Xinje XDPPro project, PLC1: XDC-32 (software 3.8.1a 2026-04-22)

PROGRAM 梯形图

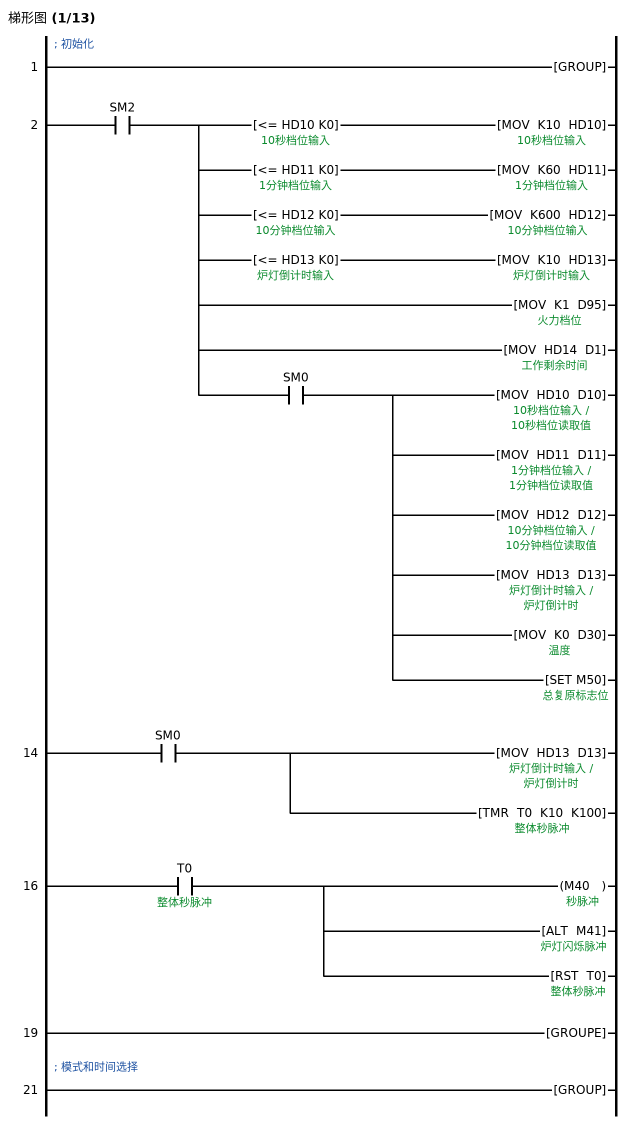
; 初始化
GROUP
LD     SM2
MPS
AND<=  HD10 K0	; 10秒档位输入
MOV    K10 HD10	; 10秒档位输入
MRD
AND<=  HD11 K0	; 1分钟档位输入
MOV    K60 HD11	; 1分钟档位输入
MRD
AND<=  HD12 K0	; 10分钟档位输入
MOV    K600 HD12	; 10分钟档位输入
MRD
AND<=  HD13 K0	; 炉灯倒计时输入
MOV    K10 HD13	; 炉灯倒计时输入
MPP
MOV    K1 D95	; 火力档位
MOV    HD14 D1	; 工作剩余时间
AND    SM0
MOV    HD10 D10	; 10秒档位输入 / 10秒档位读取值
MOV    HD11 D11	; 1分钟档位输入 / 1分钟档位读取值
MOV    HD12 D12	; 10分钟档位输入 / 10分钟档位读取值
MOV    HD13 D13	; 炉灯倒计时输入 / 炉灯倒计时
MOV    K0 D30	; 温度
SET    M50	; 总复原标志位
LD     SM0
MOV    HD13 D13	; 炉灯倒计时输入 / 炉灯倒计时
TMR    T0 K10 K100	; 整体秒脉冲
LD     T0	; 整体秒脉冲
OUT    M40	; 秒脉冲
ALT    M41	; 炉灯闪烁脉冲
RST    T0	; 整体秒脉冲
GROUPE
; 模式和时间选择
GROUP

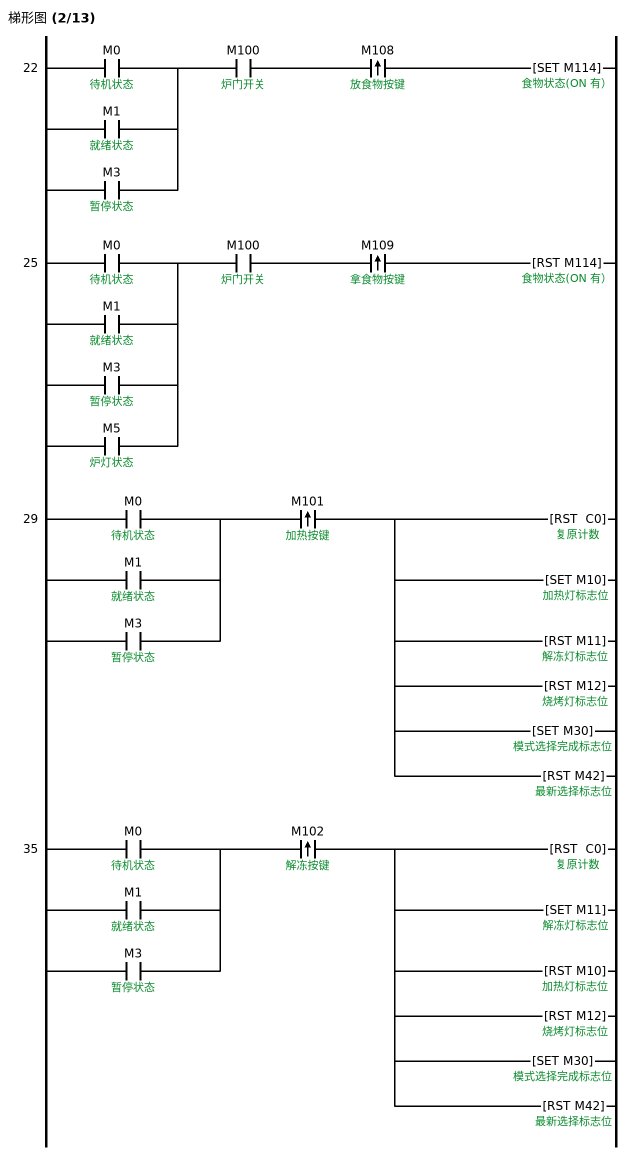
LD     M0	; 待机状态
OR     M1	; 就绪状态
OR     M3	; 暂停状态
AND    M100	; 炉门开关
ANDP   M108	; 放食物按键
SET    M114	; 食物状态(ON 有）
LD     M0	; 待机状态
OR     M1	; 就绪状态
OR     M3	; 暂停状态
OR     M5	; 炉灯状态
AND    M100	; 炉门开关
ANDP   M109	; 拿食物按键
RST    M114	; 食物状态(ON 有）
LD     M0	; 待机状态
OR     M1	; 就绪状态
OR     M3	; 暂停状态
ANDP   M101	; 加热按键
RST    C0	; 复原计数
SET    M10	; 加热灯标志位
RST    M11	; 解冻灯标志位
RST    M12	; 烧烤灯标志位
SET    M30	; 模式选择完成标志位
RST    M42	; 最新选择标志位
LD     M0	; 待机状态
OR     M1	; 就绪状态
OR     M3	; 暂停状态
ANDP   M102	; 解冻按键
RST    C0	; 复原计数
SET    M11	; 解冻灯标志位
RST    M10	; 加热灯标志位
RST    M12	; 烧烤灯标志位
SET    M30	; 模式选择完成标志位
RST    M42	; 最新选择标志位

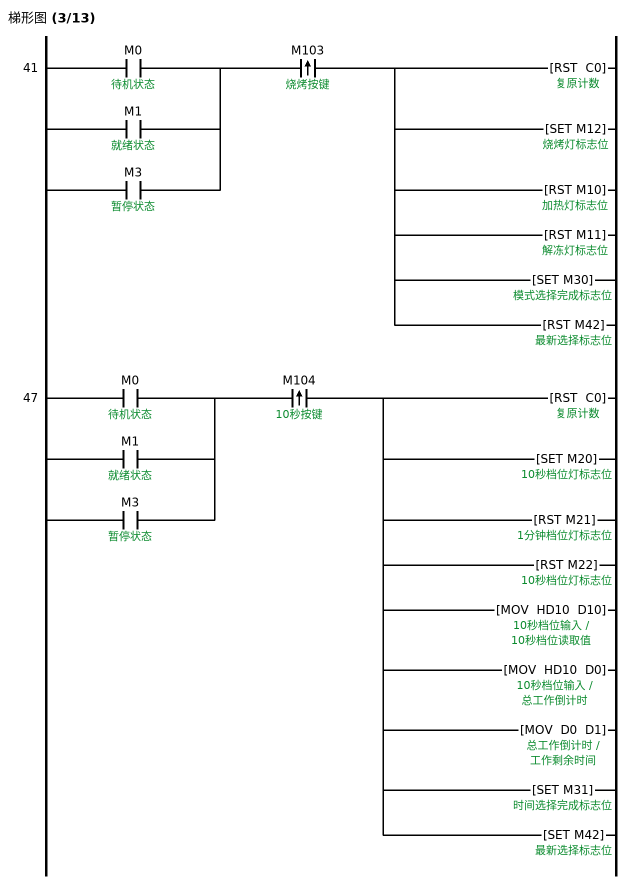
LD     M0	; 待机状态
OR     M1	; 就绪状态
OR     M3	; 暂停状态
ANDP   M103	; 烧烤按键
RST    C0	; 复原计数
SET    M12	; 烧烤灯标志位
RST    M10	; 加热灯标志位
RST    M11	; 解冻灯标志位
SET    M30	; 模式选择完成标志位
RST    M42	; 最新选择标志位
LD     M0	; 待机状态
OR     M1	; 就绪状态
OR     M3	; 暂停状态
ANDP   M104	; 10秒按键
RST    C0	; 复原计数
SET    M20	; 10秒档位灯标志位
RST    M21	; 1分钟档位灯标志位
RST    M22	; 10秒档位灯标志位
MOV    HD10 D10	; 10秒档位输入 / 10秒档位读取值
MOV    HD10 D0	; 10秒档位输入 / 总工作倒计时
MOV    D0 D1	; 总工作倒计时 / 工作剩余时间
SET    M31	; 时间选择完成标志位
SET    M42	; 最新选择标志位

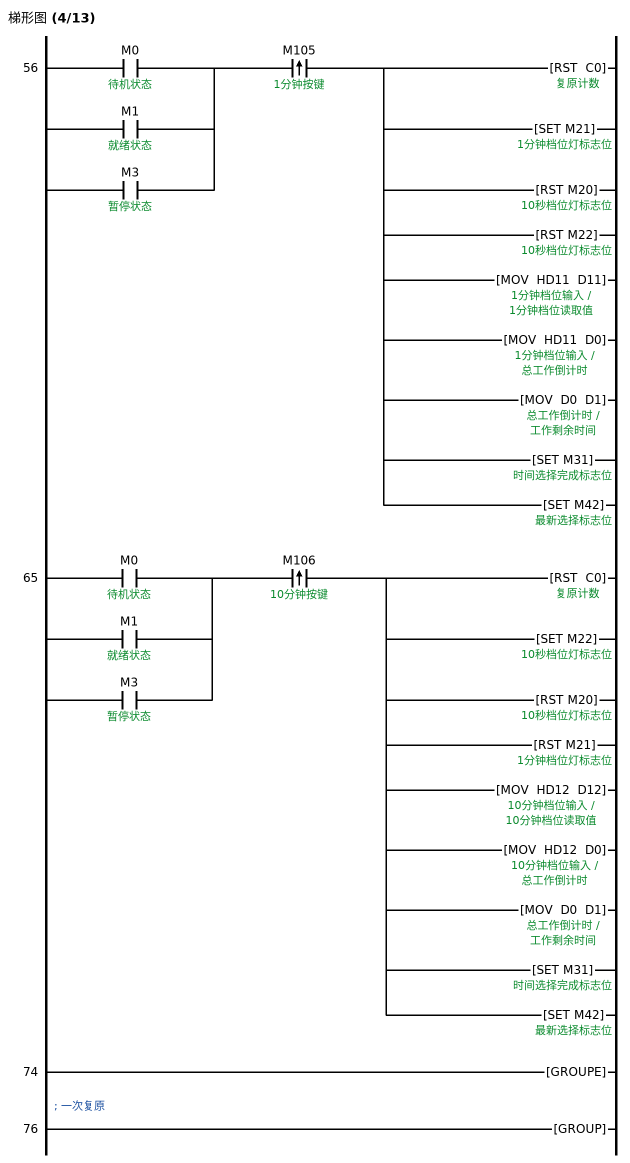
LD     M0	; 待机状态
OR     M1	; 就绪状态
OR     M3	; 暂停状态
ANDP   M105	; 1分钟按键
RST    C0	; 复原计数
SET    M21	; 1分钟档位灯标志位
RST    M20	; 10秒档位灯标志位
RST    M22	; 10秒档位灯标志位
MOV    HD11 D11	; 1分钟档位输入 / 1分钟档位读取值
MOV    HD11 D0	; 1分钟档位输入 / 总工作倒计时
MOV    D0 D1	; 总工作倒计时 / 工作剩余时间
SET    M31	; 时间选择完成标志位
SET    M42	; 最新选择标志位
LD     M0	; 待机状态
OR     M1	; 就绪状态
OR     M3	; 暂停状态
ANDP   M106	; 10分钟按键
RST    C0	; 复原计数
SET    M22	; 10秒档位灯标志位
RST    M20	; 10秒档位灯标志位
RST    M21	; 1分钟档位灯标志位
MOV    HD12 D12	; 10分钟档位输入 / 10分钟档位读取值
MOV    HD12 D0	; 10分钟档位输入 / 总工作倒计时
MOV    D0 D1	; 总工作倒计时 / 工作剩余时间
SET    M31	; 时间选择完成标志位
SET    M42	; 最新选择标志位
GROUPE
; 一次复原
GROUP

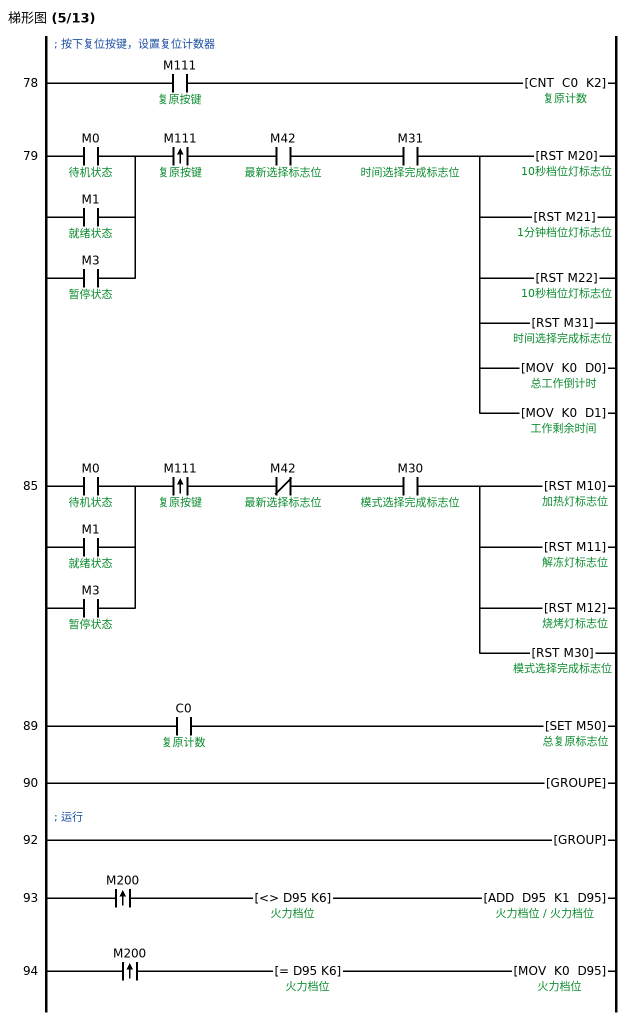
; 按下复位按键，设置复位计数器
LD     M111	; 复原按键
CNT    C0 K2	; 复原计数
LD     M0	; 待机状态
OR     M1	; 就绪状态
OR     M3	; 暂停状态
ANDP   M111	; 复原按键
AND    M42	; 最新选择标志位
AND    M31	; 时间选择完成标志位
RST    M20	; 10秒档位灯标志位
RST    M21	; 1分钟档位灯标志位
RST    M22	; 10秒档位灯标志位
RST    M31	; 时间选择完成标志位
MOV    K0 D0	; 总工作倒计时
MOV    K0 D1	; 工作剩余时间
LD     M0	; 待机状态
OR     M1	; 就绪状态
OR     M3	; 暂停状态
ANDP   M111	; 复原按键
ANI    M42	; 最新选择标志位
AND    M30	; 模式选择完成标志位
RST    M10	; 加热灯标志位
RST    M11	; 解冻灯标志位
RST    M12	; 烧烤灯标志位
RST    M30	; 模式选择完成标志位
LD     C0	; 复原计数
SET    M50	; 总复原标志位
GROUPE
; 运行
GROUP
LDP    M200
AND<>  D95 K6	; 火力档位
ADD    D95 K1 D95	; 火力档位 / 火力档位
LDP    M200
AND=   D95 K6	; 火力档位
MOV    K0 D95	; 火力档位

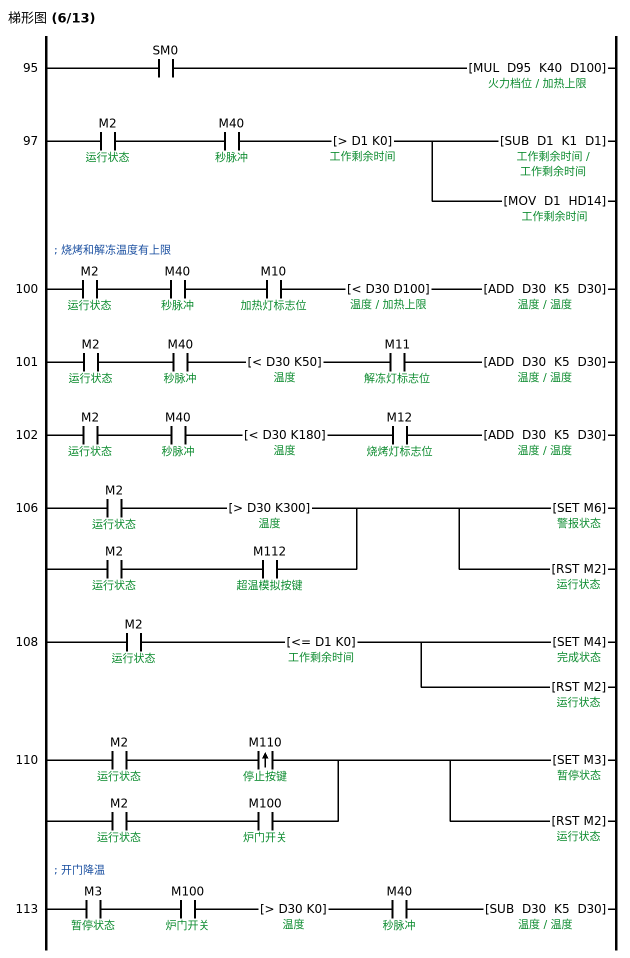
LD     SM0
MUL    D95 K40 D100	; 火力档位 / 加热上限
LD     M2	; 运行状态
AND    M40	; 秒脉冲
AND>   D1 K0	; 工作剩余时间
SUB    D1 K1 D1	; 工作剩余时间 / 工作剩余时间
MOV    D1 HD14	; 工作剩余时间
; 烧烤和解冻温度有上限
LD     M2	; 运行状态
AND    M40	; 秒脉冲
AND    M10	; 加热灯标志位
AND<   D30 D100	; 温度 / 加热上限
ADD    D30 K5 D30	; 温度 / 温度
LD     M2	; 运行状态
AND    M40	; 秒脉冲
AND<   D30 K50	; 温度
AND    M11	; 解冻灯标志位
ADD    D30 K5 D30	; 温度 / 温度
LD     M2	; 运行状态
AND    M40	; 秒脉冲
AND<   D30 K180	; 温度
AND    M12	; 烧烤灯标志位
ADD    D30 K5 D30	; 温度 / 温度
LD     M2	; 运行状态
AND>   D30 K300	; 温度
LD     M2	; 运行状态
AND    M112	; 超温模拟按键
ORB
SET    M6	; 警报状态
RST    M2	; 运行状态
LD     M2	; 运行状态
AND<=  D1 K0	; 工作剩余时间
SET    M4	; 完成状态
RST    M2	; 运行状态
LD     M2	; 运行状态
ANDP   M110	; 停止按键
LD     M2	; 运行状态
AND    M100	; 炉门开关
ORB
SET    M3	; 暂停状态
RST    M2	; 运行状态
; 开门降温
LD     M3	; 暂停状态
AND    M100	; 炉门开关
AND>   D30 K0	; 温度
AND    M40	; 秒脉冲
SUB    D30 K5 D30	; 温度 / 温度

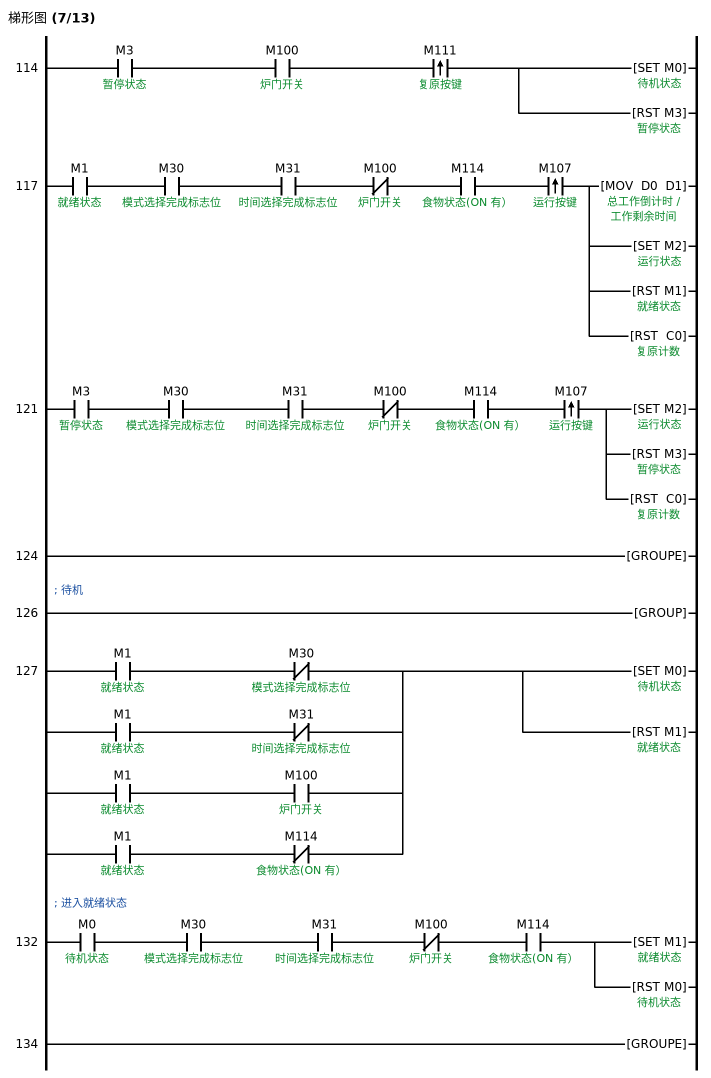
LD     M3	; 暂停状态
AND    M100	; 炉门开关
ANDP   M111	; 复原按键
SET    M0	; 待机状态
RST    M3	; 暂停状态
LD     M1	; 就绪状态
AND    M30	; 模式选择完成标志位
AND    M31	; 时间选择完成标志位
ANI    M100	; 炉门开关
AND    M114	; 食物状态(ON 有）
ANDP   M107	; 运行按键
MOV    D0 D1	; 总工作倒计时 / 工作剩余时间
SET    M2	; 运行状态
RST    M1	; 就绪状态
RST    C0	; 复原计数
LD     M3	; 暂停状态
AND    M30	; 模式选择完成标志位
AND    M31	; 时间选择完成标志位
ANI    M100	; 炉门开关
AND    M114	; 食物状态(ON 有）
ANDP   M107	; 运行按键
SET    M2	; 运行状态
RST    M3	; 暂停状态
RST    C0	; 复原计数
GROUPE
; 待机
GROUP
LD     M1	; 就绪状态
ANI    M30	; 模式选择完成标志位
LD     M1	; 就绪状态
ANI    M31	; 时间选择完成标志位
ORB
LD     M1	; 就绪状态
AND    M100	; 炉门开关
ORB
LD     M1	; 就绪状态
ANI    M114	; 食物状态(ON 有）
ORB
SET    M0	; 待机状态
RST    M1	; 就绪状态
; 进入就绪状态
LD     M0	; 待机状态
AND    M30	; 模式选择完成标志位
AND    M31	; 时间选择完成标志位
ANI    M100	; 炉门开关
AND    M114	; 食物状态(ON 有）
SET    M1	; 就绪状态
RST    M0	; 待机状态
GROUPE

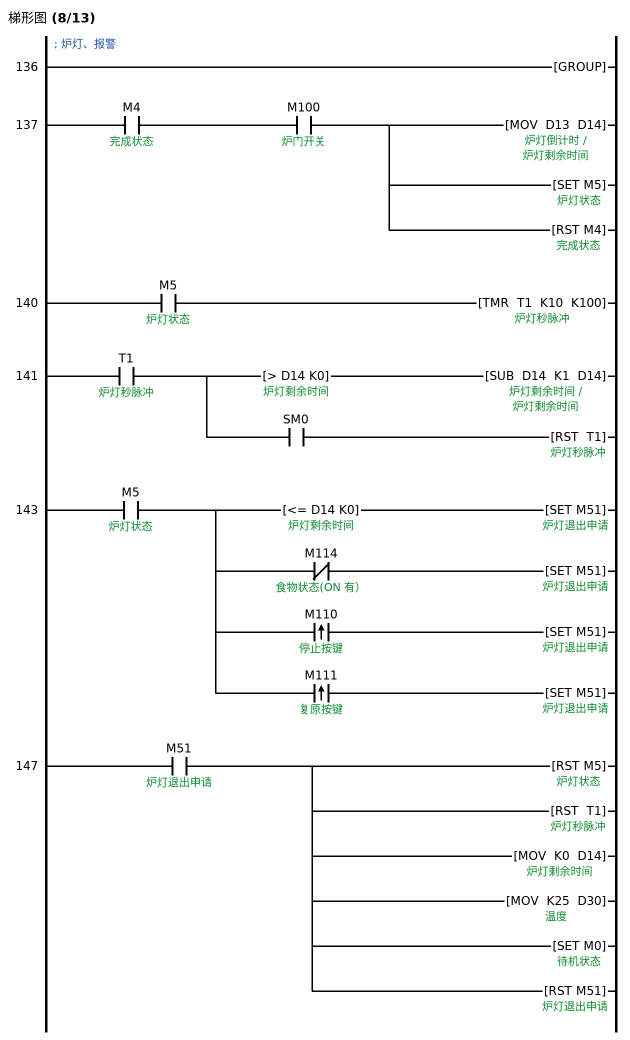
; 炉灯、报警
GROUP
LD     M4	; 完成状态
AND    M100	; 炉门开关
MOV    D13 D14	; 炉灯倒计时 / 炉灯剩余时间
SET    M5	; 炉灯状态
RST    M4	; 完成状态
LD     M5	; 炉灯状态
TMR    T1 K10 K100	; 炉灯秒脉冲
LD     T1	; 炉灯秒脉冲
MPS
AND>   D14 K0	; 炉灯剩余时间
SUB    D14 K1 D14	; 炉灯剩余时间 / 炉灯剩余时间
MPP
AND    SM0
RST    T1	; 炉灯秒脉冲
LD     M5	; 炉灯状态
MPS
AND<=  D14 K0	; 炉灯剩余时间
SET    M51	; 炉灯退出申请
MRD
ANI    M114	; 食物状态(ON 有）
SET    M51	; 炉灯退出申请
MRD
ANDP   M110	; 停止按键
SET    M51	; 炉灯退出申请
MPP
ANDP   M111	; 复原按键
SET    M51	; 炉灯退出申请
LD     M51	; 炉灯退出申请
RST    M5	; 炉灯状态
RST    T1	; 炉灯秒脉冲
MOV    K0 D14	; 炉灯剩余时间
MOV    K25 D30	; 温度
SET    M0	; 待机状态
RST    M51	; 炉灯退出申请

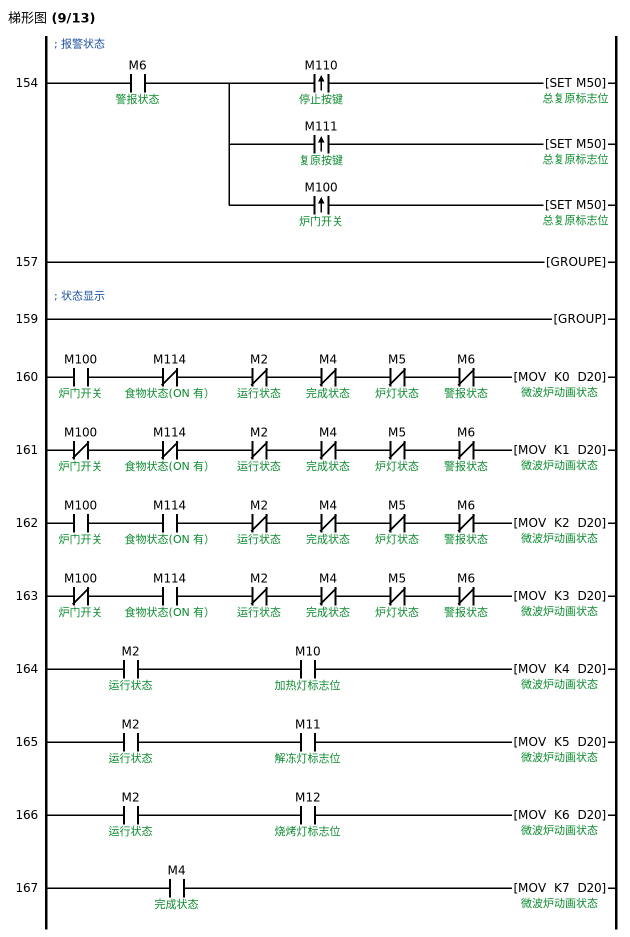
; 报警状态
LD     M6	; 警报状态
MPS
ANDP   M110	; 停止按键
SET    M50	; 总复原标志位
MRD
ANDP   M111	; 复原按键
SET    M50	; 总复原标志位
MPP
ANDP   M100	; 炉门开关
SET    M50	; 总复原标志位
GROUPE
; 状态显示
GROUP
LD     M100	; 炉门开关
ANI    M114	; 食物状态(ON 有）
ANI    M2	; 运行状态
ANI    M4	; 完成状态
ANI    M5	; 炉灯状态
ANI    M6	; 警报状态
MOV    K0 D20	; 微波炉动画状态
LDI    M100	; 炉门开关
ANI    M114	; 食物状态(ON 有）
ANI    M2	; 运行状态
ANI    M4	; 完成状态
ANI    M5	; 炉灯状态
ANI    M6	; 警报状态
MOV    K1 D20	; 微波炉动画状态
LD     M100	; 炉门开关
AND    M114	; 食物状态(ON 有）
ANI    M2	; 运行状态
ANI    M4	; 完成状态
ANI    M5	; 炉灯状态
ANI    M6	; 警报状态
MOV    K2 D20	; 微波炉动画状态
LDI    M100	; 炉门开关
AND    M114	; 食物状态(ON 有）
ANI    M2	; 运行状态
ANI    M4	; 完成状态
ANI    M5	; 炉灯状态
ANI    M6	; 警报状态
MOV    K3 D20	; 微波炉动画状态
LD     M2	; 运行状态
AND    M10	; 加热灯标志位
MOV    K4 D20	; 微波炉动画状态
LD     M2	; 运行状态
AND    M11	; 解冻灯标志位
MOV    K5 D20	; 微波炉动画状态
LD     M2	; 运行状态
AND    M12	; 烧烤灯标志位
MOV    K6 D20	; 微波炉动画状态
LD     M4	; 完成状态
MOV    K7 D20	; 微波炉动画状态

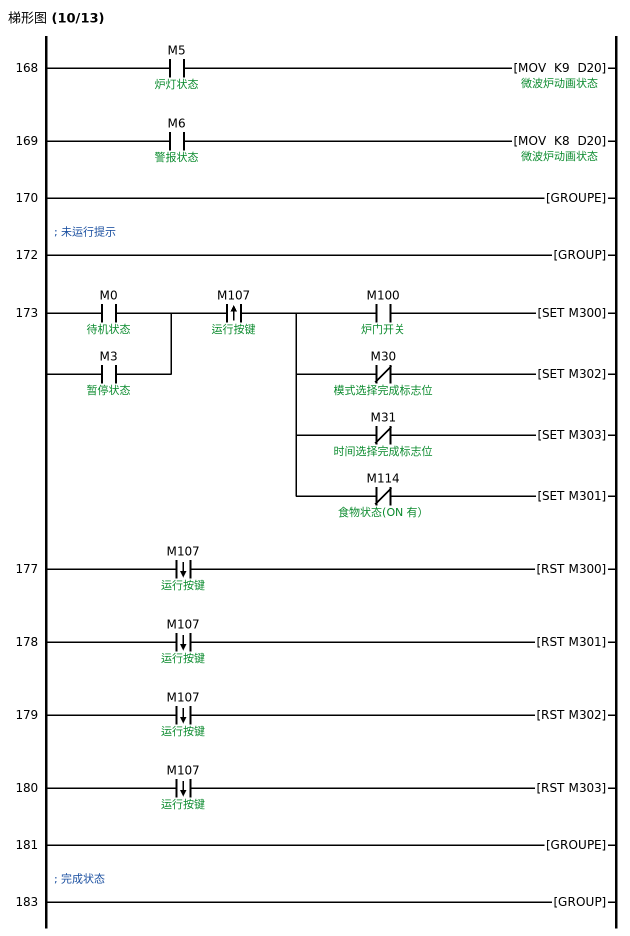
LD     M5	; 炉灯状态
MOV    K9 D20	; 微波炉动画状态
LD     M6	; 警报状态
MOV    K8 D20	; 微波炉动画状态
GROUPE
; 未运行提示
GROUP
LD     M0	; 待机状态
OR     M3	; 暂停状态
ANDP   M107	; 运行按键
MPS
AND    M100	; 炉门开关
SET    M300
MRD
ANI    M30	; 模式选择完成标志位
SET    M302
MRD
ANI    M31	; 时间选择完成标志位
SET    M303
MPP
ANI    M114	; 食物状态(ON 有）
SET    M301
LDF    M107	; 运行按键
RST    M300
LDF    M107	; 运行按键
RST    M301
LDF    M107	; 运行按键
RST    M302
LDF    M107	; 运行按键
RST    M303
GROUPE
; 完成状态
GROUP

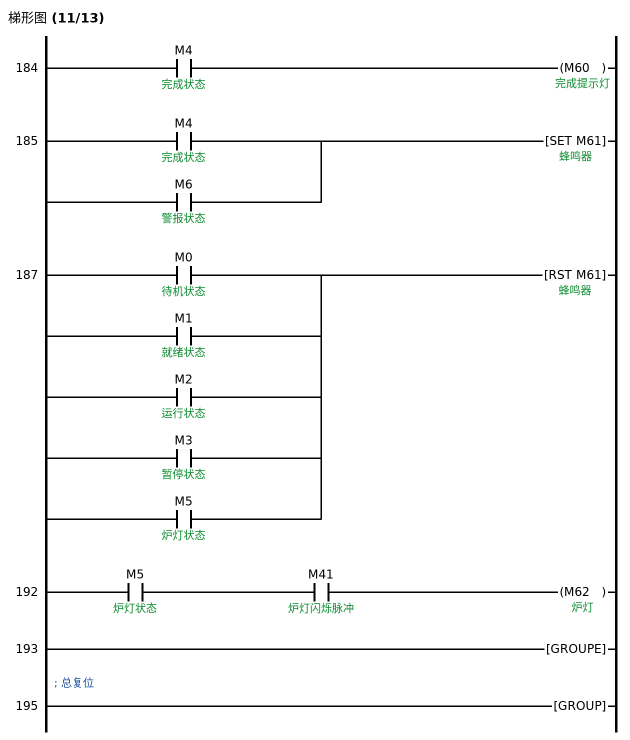
LD     M4	; 完成状态
OUT    M60	; 完成提示灯
LD     M4	; 完成状态
OR     M6	; 警报状态
SET    M61	; 蜂鸣器
LD     M0	; 待机状态
OR     M1	; 就绪状态
OR     M2	; 运行状态
OR     M3	; 暂停状态
OR     M5	; 炉灯状态
RST    M61	; 蜂鸣器
LD     M5	; 炉灯状态
AND    M41	; 炉灯闪烁脉冲
OUT    M62	; 炉灯
GROUPE
; 总复位
GROUP

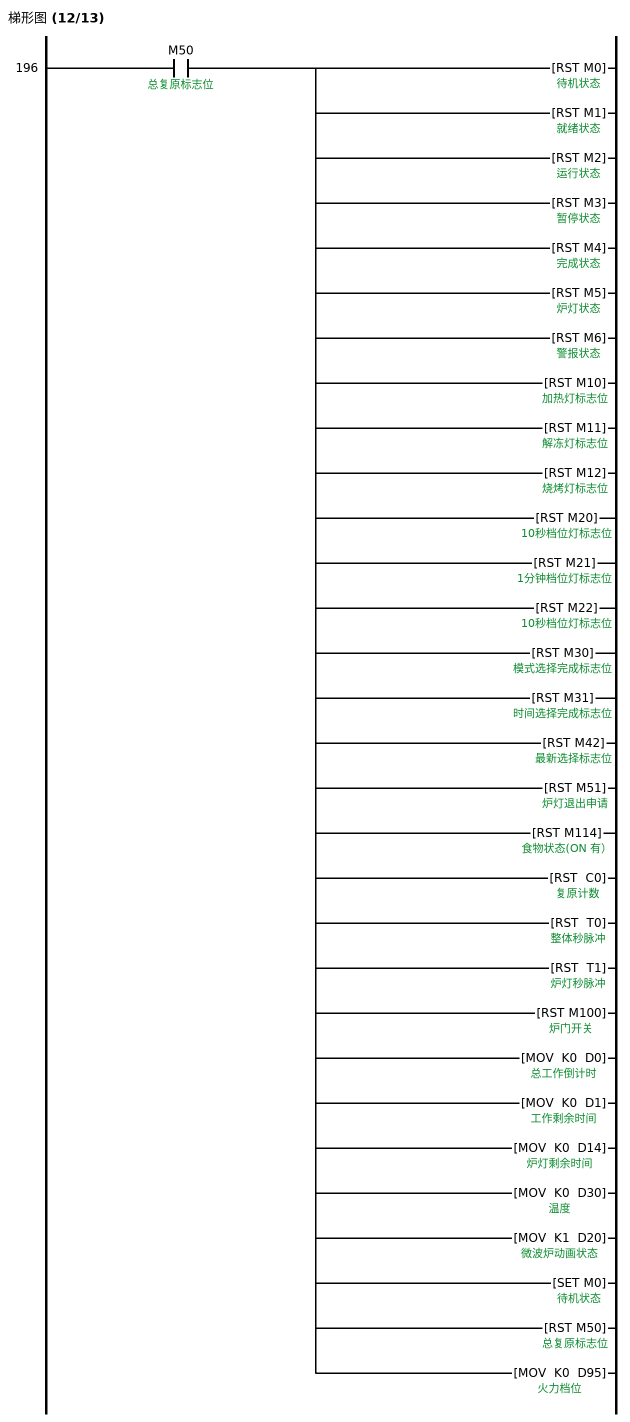
LD     M50	; 总复原标志位
RST    M0	; 待机状态
RST    M1	; 就绪状态
RST    M2	; 运行状态
RST    M3	; 暂停状态
RST    M4	; 完成状态
RST    M5	; 炉灯状态
RST    M6	; 警报状态
RST    M10	; 加热灯标志位
RST    M11	; 解冻灯标志位
RST    M12	; 烧烤灯标志位
RST    M20	; 10秒档位灯标志位
RST    M21	; 1分钟档位灯标志位
RST    M22	; 10秒档位灯标志位
RST    M30	; 模式选择完成标志位
RST    M31	; 时间选择完成标志位
RST    M42	; 最新选择标志位
RST    M51	; 炉灯退出申请
RST    M114	; 食物状态(ON 有）
RST    C0	; 复原计数
RST    T0	; 整体秒脉冲
RST    T1	; 炉灯秒脉冲
RST    M100	; 炉门开关
MOV    K0 D0	; 总工作倒计时
MOV    K0 D1	; 工作剩余时间
MOV    K0 D14	; 炉灯剩余时间
MOV    K0 D30	; 温度
MOV    K1 D20	; 微波炉动画状态
SET    M0	; 待机状态
RST    M50	; 总复原标志位
MOV    K0 D95	; 火力档位

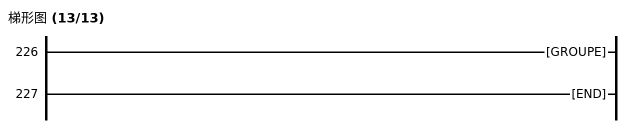
GROUPE
END